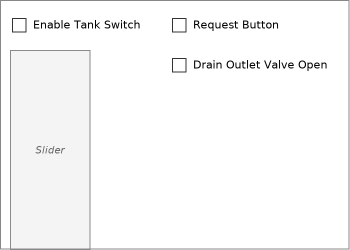
VISUALIZATION Vi_Sim_Tank  // 350x250
VAR_IN_OUT
	obj			: Tank;
	obj2		: Outlet;
END_VAR
    Checkbox (10,10 160x30), "Enable Tank Switch", variable: obj.bEnable
    Slider (10,50 80x200), variable: obj.fLevel, scale 0..2
    Checkbox (170,50 180x30), "Drain Outlet Valve Open", variable: obj2.bDrainValveOpen
    Checkbox (170,10 180x30), "Request Button", variable: obj2.bRequestButton
END_VISUALIZATION

(* stored: Version 1.1.0.1
   Visu Vi_Sim_Tank: Id {0e800f35-bca0-47d3-b83a-0eec2e426a21} *)
